// TIA Portal project "Filling Tank_V17" (V17)
// Vorlageprojekt für das Buch mit Zielsystem S7-1200

(* hardware
DEVICE "S7-1200-Station_1"  S7-1200 Station
   slot 0: "Baugruppenträger_0"  Rack  V1.0
   slot 1: "PLC_1"  CPU 1211C DC/DC/DC  6ES7 211-1AE40-0XB0  V4.1
DEVICE "HMI_1"  TP700 Comfort
   slot 0: "HMI_1"  TP700 Comfort  6AV2 124-0GC01-0AX0  15.0.0.0
   slot 1: "HMI_RT_1"  TP700 Comfort  6AV2 124-0GC01-0AX0  15.0.0.0
   slot 5: "HMI_1.IE_CP_1"  PROFINET Interface  15.0.0.0
      slot 1: "PROFINET Interface_1"  PROFINET Interface
         slot 1: "Port_1"  Port
         slot 2: "Port_2"  Port
   slot 7: "HMI_1.MPI/DP_CP_1"  MPI/DP Interface  15.0.0.0
*)

// ===== PLC "PLC_1"  CPU 1211C DC/DC/DC =====

VAR_GLOBAL   // PLC tag table "Standard-Variablentabelle"
   "start" AT %I0.0 : Bool;
   "stop" AT %I0.1 : Bool;
   "drain" AT %I0.2 : Bool;
   "levelMeter" AT %ID30 : Real;
   "SetPoint" AT %ID38 : Real;
   "FillValve" AT %QD30 : Real;
   "DissValve" AT %QD34 : Real;
   "SetPointDisplay" AT %QD38 : DInt;
   "LevelDisplay" AT %QD42 : DInt;
   "ErrorDisplay" AT %QD46 : Real;
   "Tag_1" AT %M0.0 : Bool;
   "Tag_2" AT %MD100 : Real;
   "scaledlevel" AT %MW2 : Int;
   "setscaled" AT %MW12 : Int;
   "Tag_3" AT %M2.2 : Bool;
END_VAR

DATA_BLOCK "PI_DB"   // DB3
{ S7_Optimized_Access := 'TRUE' }
VERSION : 0.1
// stored: InstanceOfName PID
"PID"
BEGIN
END_DATA_BLOCK

DATA_BLOCK "hmi"   // DB5
{ S7_Optimized_Access := 'TRUE' }
VERSION : 0.1
   VAR
      startfromhmi : Bool;
   END_VAR
BEGIN
END_DATA_BLOCK

DATA_BLOCK "PID_DB"   // DB6
{ S7_Optimized_Access := 'TRUE' }
VERSION : 0.1
// stored: InstanceOfName PID
"PID"
BEGIN
END_DATA_BLOCK

FUNCTION_BLOCK "PID"   // FB1, SCL
{ S7_Optimized_Access := 'TRUE' }
VERSION : 0.1
   VAR_INPUT
      ki : Real := 0.002;
      kp : Real := 11.0;
      kd : Real;
      level : Real;
      setpoint : Real;
      drain : Bool;
      "full drain" : Bool;
      emergency : Bool;
   END_VAR
   VAR_OUTPUT
      filling : Real;
      draining : Real;
      errordisplay : Real;
      setpointdisplay : DInt;
      leveldisplay : DInt;
   END_VAR
   VAR
      integralop : Real;
      oldintegral : Real;
      err2 : Real;
   END_VAR
   VAR_TEMP
      error : Real;
      u : Real;
      temp : DInt;
   END_VAR
BEGIN

   #errordisplay := ABS(#setpoint - #level);

   //display setpoint to 100%
   #setpointdisplay := REAL_TO_DINT(#setpoint*10.0);
   //



   //display level to 100%
   #leveldisplay :=REAL_TO_DINT( #level*10.0);
   //
   #temp := REAL_TO_DINT(#kp);

   #error := #setpoint - #level;

   #integralop := #integralop + #error; //sums all the past errors to present error
   #u := (#error * #kp) + (#integralop * (#ki / 10)) + (#kd * (#err2 - #error));
   #filling := #u;
   #draining := -#u;


   //if error always goes up the filling will always goes up
   //and it will be more that 100% .but the valve can go only to 100% open
   //so if it goes up.we stop the valve at 10 and  stabilized the integral
   IF (#filling > 10.0) THEN
       #integralop := #oldintegral;
       #filling := 10.0;
   END_IF;
   //same thing but for values under 0
   IF (#filling < 0.0) THEN
       #integralop := #oldintegral;
       #filling := 0.0;
   END_IF;
   IF (#draining > 10.0) THEN
       #integralop := #oldintegral;
       #draining := 10.0;
   END_IF;

   IF (#draining < 0.0) THEN
       #integralop := #oldintegral;
       #draining := 0.0;
   END_IF;

   #oldintegral := #integralop; //past error sum
   #err2 := #error;//past error

   IF #drain THEN
       #draining := 10.0;

   END_IF;

   IF #"full drain" THEN
       #draining := 10.0;
       #filling := 0;
   END_IF;
   IF #emergency THEN
       #draining := 0;
       #filling := 0;

   END_IF;
END_FUNCTION_BLOCK

FUNCTION "MHJ-PLC-Lab-Function-S71200" : Void   // FC9000, SCL
{ S7_Optimized_Access := 'TRUE' }
VERSION : 0.1
   VAR_TEMP
      rdTimeReturn : Int;
      outputTime : DTL;
      SyncVal : Byte;
      forVal : Int;
      forVal_2 : Int;
      Value : Byte;
   END_VAR
   VAR CONSTANT
      CompVal : Byte := 16#34;
      Value_01 : Byte := 16#11;
      Value_01_DW : DWord := 16#A165_D992;
      Value_02_DW : DWord := 16#58BE_4401;
   END_VAR
BEGIN

   #Value:=PEEK(area := 16#82,
        dbNumber := 0,
        byteOffset := 511);
   #Value := #Value + 1;

   POKE(area := 16#82,
        dbNumber := 0,
        byteOffset := 511,
        value := #Value);

   POKE(area:=16#81,
        dbNumber:=0,
        byteOffset:=1016,
        value:=#Value_01_DW);
   POKE(area := 16#81,
        dbNumber := 0,
        byteOffset := 1020,
        value := #Value_02_DW);

   POKE(area := 16#81,
        dbNumber := 0,
        byteOffset := 511,
        value := B#16#00);

   FOR #forVal := 0 TO 120 DO
       FOR #forVal_2:=0 TO 10 DO
           #rdTimeReturn:=RD_SYS_T(#outputTime);
           #rdTimeReturn := WR_SYS_T(#outputTime);
           #rdTimeReturn := RD_SYS_T(#outputTime);
           #rdTimeReturn := WR_SYS_T(#outputTime);
       END_FOR;
       #SyncVal:= PEEK(area := 16#81,
                      dbNumber := 0,
                      byteOffset := 511);
       IF #SyncVal = #CompVal THEN
          GOTO M_1;
       END_IF;
   END_FOR;
   RETURN;

   M_1:
   POKE(area := 16#81,
        dbNumber := 0,
        byteOffset := 511,
        value := B#16#0);
END_FUNCTION

ORGANIZATION_BLOCK "Main"   // OB1, LAD, ProgramCycle
TITLE = "Main Program Sweep (Cycle)"
{ S7_Optimized_Access := 'TRUE' }
VERSION : 0.1
   VAR_INPUT
      Initial_Call : Bool;   // Initial call of this OB
      Remanence : Bool;   // =True, if remanent data are available
   END_VAR
   VAR_TEMP
      norm3 : Real;
   END_VAR
BEGIN

REGION Network 1: Konnektierungsbaustein für PLC-Lab / FOR FACTORY I/O
   // Im Netzwerk 1 wird der Konnektierungsbaustein für PLC-Lab aufgerufen.
   // Dieser Aufruf darf nicht entfernt werden!
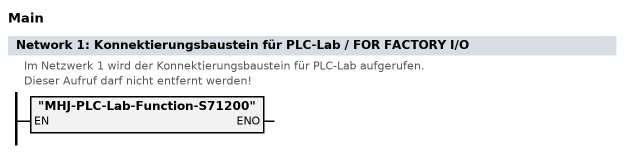
   RUNG wire#powerrail
      "MHJ-PLC-Lab-Function-S71200"()
   END_RUNG
   // the same network as SCL:
   "MHJ-PLC-Lab-Function-S71200"();
END_REGION
END_ORGANIZATION_BLOCK

ORGANIZATION_BLOCK "Cyclic interrupt"   // OB30, LAD, CyclicInterrupt
{ S7_Optimized_Access := 'TRUE' }
VERSION : 0.1
   VAR_INPUT
      Initial_Call : Bool;   // Initial call of this OB
      Event_Count : Int;   // Events discarded
   END_VAR
BEGIN

REGION Network 1
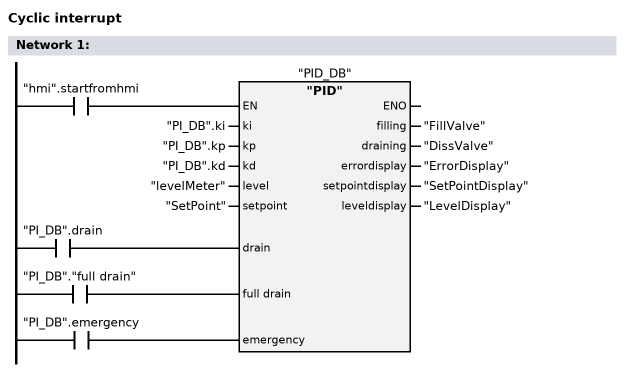
   RUNG wire#powerrail
      Contact( "hmi".startfromhmi )
      "PID_DB"(drain := wire#w1, "full drain" := wire#w2, emergency := wire#w3, ki := "PI_DB".ki, kp := "PI_DB".kp, kd := "PI_DB".kd, level := "levelMeter", setpoint := "SetPoint", filling => "FillValve", draining => "DissValve", errordisplay => "ErrorDisplay", setpointdisplay => "SetPointDisplay", leveldisplay => "LevelDisplay")
   END_RUNG
   RUNG wire#powerrail
      Contact( "PI_DB".drain )
   END_RUNG wire#w1
   RUNG wire#powerrail
      Contact( "PI_DB"."full drain" )
   END_RUNG wire#w2
   RUNG wire#powerrail
      Contact( "PI_DB".emergency )
   END_RUNG wire#w3
   // the same network as SCL:
   IF "hmi".startfromhmi THEN
       "PID_DB"(ki := "PI_DB".ki,   // "PID"
                kp := "PI_DB".kp,
                kd := "PI_DB".kd,
                level := "levelMeter",
                setpoint := "SetPoint",
                drain := "PI_DB".drain,
                "full drain" := "PI_DB"."full drain",
                emergency := "PI_DB".emergency,
                filling => "FillValve",
                draining => "DissValve",
                errordisplay => "ErrorDisplay",
                setpointdisplay => "SetPointDisplay",
                leveldisplay => "LevelDisplay");
   END_IF;
END_REGION

REGION Network 2 (SCL): TO BE SURE THAT KP ON PID WILL BE ALWAYS BIGGER THAN 1
   IF "PI_DB".kp < 1 THEN
       "PI_DB".kp := 1;
   END_IF;
END_REGION
END_ORGANIZATION_BLOCK

(* ===== HMI "HMI_RT_1" =====
system functions are stored by id; their names below are inferred from use
connection "HMI_Connection_1": ETHERNET, S7_1200_OMS

HMI tags "Default tag table"
   "Tag_ScreenNumber" : UInt, internal
   "PI_DB_ki" : Real = PLC PI_DB.ki, 1 s
   "PI_DB_kp" : Real = PLC PI_DB.kp, 1 s
   "PI_DB_kd" : Real = PLC PI_DB.kd, 1 s
   "PI_DB_errordisplay" : Real = PLC PI_DB.errordisplay, 1 s
   "PI_DB_drain" : Bool = PLC PI_DB.drain, 1 s
   "start" : Bool = PLC start AT %I0.0, 1 s
   "hmi_startfromhmi" : Bool = PLC hmi.startfromhmi, 1 s
   "PI_DB_leveldisplay" : DInt = PLC PI_DB.leveldisplay, 1 s
   "PI_DB_setpoint" : Real = PLC PI_DB.setpoint, 1 s
   "PI_DB_full drain" : Bool = PLC PI_DB."full drain", 1 s
   "PI_DB_emergency" : Bool = PLC PI_DB.emergency, 1 s
   "PID_DB_leveldisplay" : DInt = PLC PID_DB.leveldisplay, 1 s
   "PID_DB_errordisplay" : Real = PLC PID_DB.errordisplay, 1 s
   "PID_DB_setpointdisplay" : DInt = PLC PID_DB.setpointdisplay, 1 s
   "check" : Int, internal

analog alarms
   1: 'Kd maybe cause troumble on the control', class Warnings, trigger "PI_DB_kd"
      on Going: function_b9b71300("check", 1)
      on Coming: function_dd21b452("check", 1)
   2: 'Ki has a high value', class Warnings, trigger "PI_DB_ki"
      on Coming: function_dd21b452("check", 1)
      on Going: function_b9b71300("check", 1)

screen "Root screen" 800x420, template "Template_1"
   on GenerateScreen: SetTag("Tag_ScreenNumber", 1); function_f23ef4c9()
   IOField "I/O field_4" at 13,300 size 120x32; FormatPattern s999.999
      ProcessValue <- "PID_DB_errordisplay"
   TextField "Text field_4" at 14,268 size 128x26; Text 'Error Display'
   Button "Button_1" at 15,75 size 154x47; TextOff 'DRAIN'
      on Press: function_b14e0dd5("PI_DB_drain", 0)
   Button "Button_2" at 14,13 size 154x47; TextOff 'START'
      on Release: SetBit("hmi_startfromhmi")
   GraphicView "Graphic view_1" at 587,8 size 178x273; Picture "Graphic_5"
   Bar "Bar_1" at 589,23 size 174x139; MinimumValue 0; MaximumValue 100
      ProcessValue <- "PID_DB_leveldisplay"
   Switch "Switch_1" at 243,68 size 154x54; CaptionText 'FULL DRAIN'; TextOff 'OFF'; TextOn 'ON'
      ProcessValue <- "PI_DB_full drain"
   Switch "Switch_2" at 215,0 size 280x64; CaptionText 'EMERGENCY STOP'; TextOff 'OFF'; TextOn 'ON'
      ProcessValue <- "PI_DB_emergency"
   TextField "Text field_1" at 533,310 size 267x42; Text 'You Need to be Admin to change the Kp,Ki,Kd value'
   GraphicView "Graphic view_2" at 480,314 size 46x38; Picture "Graphic_8"
   IOField "I/O field_1" at 15,170 size 120x32; FormatPattern s9999999
      ProcessValue <- "PID_DB_setpointdisplay"
   TextField "Text field_2" at 8,144 size 201x26; Text 'SetPoint Display(%)'
   IOField "I/O field_5" at 14,236 size 120x32; FormatPattern s9999999
      ProcessValue <- "PID_DB_leveldisplay"
   TextField "Text field_6" at 13,206 size 196x29; Text 'Level Display(%)'
   IOField "I/O field_2" at 262,328 size 96x32; FormatPattern 99.9999
      ProcessValue <- "PI_DB_ki"
   IOField "I/O field_3" at 156,329 size 96x32
      ProcessValue <- "PI_DB_kp"
   IOField "I/O field_6" at 368,329 size 96x32
      ProcessValue <- "PI_DB_kd"
   TextField "Text field_3" at 181,306 size 28x23; Text 'Kp'
   TextField "Text field_5" at 292,306 size 23x23; Text 'Ki'
   TextField "Text field_7" at 397,305 size 28x23; Text 'Kd'

Template "Template_1" 800x420
   Button "Exit" at 720,360 size 78x58; TextOff 'Exit'; PictureOff "ExitRuntime_TP700_Comfort_TR"; PictureOn "ExitRuntime_TP700_Comfort_TR"
      on Release: StopRuntime(0)
   Button "Template_Button" at 640,360 size 78x58; TextOff 'Text'
   Button "Template_Button_1" at 560,360 size 78x58; TextOff 'Text'
   Button "Template_Button_2" at 480,360 size 78x58; TextOff 'Text'
   Button "Template_Button_3" at 400,360 size 78x58; TextOff 'Text'
   Button "Template_Button_4" at 321,360 size 78x58; TextOff 'Text'
   Button "Template_Button_5" at 241,360 size 78x58; TextOff 'Text'
   Button "Template_Button_6" at 161,360 size 78x58; TextOff 'Error screen'
      on Click: ActivateScreen("Error screen", 0)
      Appearance <- "check"
   Button "Template_Button_7" at 81,360 size 78x58; TextOff 'ADMIN SCREEN'; PictureOff "NavigateHome_TP700_Comfort_TR"; Authorization "Admin screen"
      on Release: ActivateScreen("Admin Screen", 0)
   Button "Start screen" at 1,360 size 78x58; TextOff 'Start screen'; PictureOff "NavigateHome_TP700_Comfort_TR"; PictureOn "NavigateHome_TP700_Comfort_TR"
      on Release: ActivateScreen("Root screen", 0)

screen "Admin Screen" 800x420, template "Template_1"
   TextField "Text field_1" at 309,124 size 144x23; Text 'ADMIN SCREEN'
   Group "Group" at 6,96 size 161x163
   Group "Group_1" at 5,273 size 483x44; Picture "Graphic_2"
   Button "Button_3" at 639,305 size 154x47; TextOff 'STOP PID'
      on Release: ResetBit("hmi_startfromhmi")
   IOField "I/O field_1" at 47,154 size 120x47; FormatPattern 999999.999
      ProcessValue <- "PI_DB_ki"
   TextField "Text field_2" at 6,161 size 28x29; Text 'Ki'
   IOField "I/O field_2" at 47,96 size 120x47; FormatPattern 999999.999
      ProcessValue <- "PI_DB_kp"
   IOField "I/O field_3" at 47,212 size 120x47; FormatPattern 999999.999
      ProcessValue <- "PI_DB_kd"
   TextField "Text field_3" at 6,220 size 35x29; Text 'Kd'
   TextField "Text field_4" at 6,99 size 35x29; Text 'Kp'
   GraphicView "Graphic view_2" at 5,273 size 36x30; Picture "Graphic_2"
   TextField "Text field_5" at 28,279 size 460x38; Text ': Recommended (and starting) values for the level control Kp=11 ,Ki=0.002,kd=0.0'

screen "Error screen" 800x420, template "Template_1"
   AlarmView "Alarm view_1" at 87,17 size 645x322
*)